INTERFACE I_MoveCommand EXTENDS I_Command

END_INTERFACE

(* stored: Version 1.1.0.1, ProductVersion 3.1.4024.12
   Itf I_MoveCommand: Id {ace235f2-e3c9-4384-9979-8089e1813370} *)
